// TIA Portal V19 export
DATA_BLOCK "PPrgArchive3"   // DB520
// stored: IsOnlyStoredInLoadMemory true, MemoryReserve 0, Namespace G
   VAR RETAIN
      PRG : Array[201..300] of "PPrg_Data";
   END_VAR
BEGIN
END_DATA_BLOCK
